FUNCTION_BLOCK Resetting_State_Sample  IMPLEMENTS ITF_State
VAR_INPUT
END_VAR
VAR_OUTPUT
END_VAR
VAR
	pPML_Base : POINTER TO PML_StatePattern_Base;
	_stateMachine : IPmlStateMachine;
	bResetComplete : BOOL;
END_VAR

METHOD Cycle : BOOL
VAR_INPUT
END_VAR
IF bResetComplete THEN
	_stateMachine.SetStateComplete();
	pPML_Base^.SetState(pPML_Base^.idle);
END_IF
END_METHOD

METHOD FB_init : BOOL
VAR_INPUT
	bInitRetains : BOOL; // if TRUE, the retain variables are initialized (warm start / cold start)
	bInCopyCode : BOOL;  // if TRUE, the instance afterwards gets moved into the copy code (online change)
	pPML_Base : POINTER TO PML_StatePattern_Base;
	statemachine : IPmlStateMachine;
END_VAR
_stateMachine := statemachine;
THIS^.pPML_Base := pPML_Base;
END_METHOD

END_FUNCTION_BLOCK

(* stored: Version 1.1.0.1, ProductVersion 3.1.4024.11
   POU Resetting_State_Sample: Id {a55d4d71-4945-4a20-a665-8ca399172363}, SpecialFunc None
   Method Cycle: Id {882ac881-ce51-4945-bc3b-0233053efdf6}
   Method FB_init: Id {b4c451d4-f077-4abd-bb7b-0ca54e25926c} *)
